TYPE VFDI EXTENDS MotorI :
STRUCT
	InputFreq : INT;
	RampRate : INT;
	FreqMaxSignal : INT;
END_STRUCT
END_TYPE

(* stored: Version 1.1.0.1, ProductVersion 3.1.4024.12
   DUT VFDI: Id {24a5297a-8ddf-4152-973c-2fa5840a1f61} *)
